// TIA Portal V19 export
FUNCTION "Manager" : Void   // FC201, LAD
{ S7_Optimized_Access := 'TRUE' }
AUTHOR : CH
FAMILY : Aktina
NAME : PROCESS
// stored: AutoNumber false, SetENOAutomatically false
   VAR CONSTANT
      maxVol : Real := 45359.24;
   END_VAR
BEGIN

REGION Network 1 (SCL): Tank mbar to vol
END_REGION

REGION Network 2 (SCL): // Process Function
END_REGION
END_FUNCTION
